TYPE ControlStewart :
STRUCT
	surge : REAL := 0.0;
	sway : REAL := 0.0;
	heave : REAL := 0.0;
	phi : REAL := 0.0;
	theta : REAL := 0.0;
	psi : REAL := 0.0;
END_STRUCT
END_TYPE

(* stored: Version 1.1.0.1, ProductVersion 3.1.4020.12
   DUT ControlStewart: Id {82a91836-017b-4067-ba62-e78e727836e4} *)
